// SIMATIC S7-200 SMART project (STEP 7-Micro/WIN SMART), CPU SR40

ORGANIZATION_BLOCK 主程序:OB1
TITLE=
BEGIN
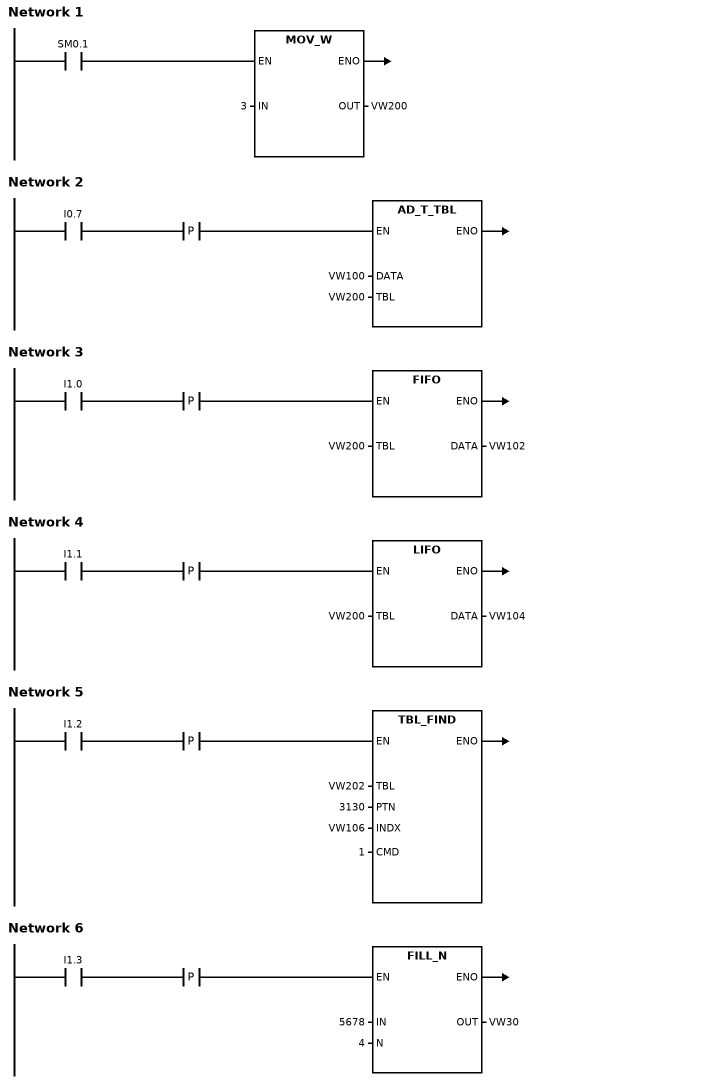
Network 1
LD     SM0.1
MOVW   3, VW200
Network 2
LD     I0.7
EU
ATT    VW100, VW200
Network 3
LD     I1.0
EU
FIFO   VW200, VW102
Network 4
LD     I1.1
EU
LIFO   VW200, VW104
Network 5
// (network saved uncompiled; LAD cells follow)
// row 0: c0 -| |- I1.2  c1 -|P|-  c2 --  c3 [TBL_FIND EN:=power@row0, TBL:=VW202, PTN:=3130, INDX:=VW106, CMD:=1, ENO=>power]  c4 ->
// row 1: c3 [box]
// row 2: c3 [box]
Network 6
// (network saved uncompiled; LAD cells follow)
// row 0: c0 -| |- I1.3  c1 -|P|-  c2 --  c3 [FILL_N EN:=power@row0, IN:=5678, N:=4, ENO=>power, OUT=>VW30]  c4 ->
// row 1: c3 [box]
END_ORGANIZATION_BLOCK
